FUNCTION_BLOCK EQ_StopperArm (* Servo that places the stopper; 0..180 degrees (outer home 120, inner 1), no feedback; equipment IO: owns its IO points, writes the output values its holder sends, reads its inputs every cycle and reports changes *)
  (* Standard: 61499-2 *)
  (* Version 0.1, 2026-09-28, Project contributors, AAU Smart Production Lab *)
  PACKAGE stoppering;
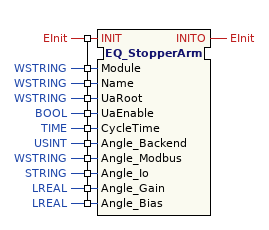
  EVENT_INPUT
    INIT : EInit WITH Module, Name, UaRoot, UaEnable, CycleTime, Angle_Backend, Angle_Modbus, Angle_Io, Angle_Gain, Angle_Bias;
  END_EVENT
  EVENT_OUTPUT
    INITO : EInit;
  END_EVENT
  VAR_INPUT
    Module : WSTRING;
    Name : WSTRING := "StopperArm";
    UaRoot : WSTRING;
    UaEnable : BOOL;
    CycleTime : TIME := T#50ms;
    Angle_Backend : USINT := 2;
    Angle_Modbus : WSTRING;
    Angle_Io : STRING;
    Angle_Gain : LREAL := 36.408;
    Angle_Bias : LREAL := 1638.4;
  END_VAR
  (* Group Core: One holder at a time, break before make, all off on release or abort; scanned every CycleTime *)
  (* Group Channels: Local channels to and from the skills (cmd, release, state), the module's state, and the inputs over OPC UA *)
  (* Group Outputs: The equipment's actuators: written on a change and every cycle, one block per IO point *)
  FBS
    Logic : stoppering::EL_StopperArm; {SET_ATTRIBUTE(GroupName, Core)}
    Cycle : iec61499::events::E_CYCLE; {SET_ATTRIBUTE(GroupName, Core)}
    Mode : modlib::MOD_StateView; {SET_ATTRIBUTE(GroupName, Channels)}
    SubCmd : iec61499::net::SUBSCRIBE_4(QI := TRUE); {SET_ATTRIBUTE(GroupName, Channels)}
    SubRelease : iec61499::net::SUBSCRIBE_1(QI := TRUE); {SET_ATTRIBUTE(GroupName, Channels)}
    PubState : iec61499::net::PUBLISH_1(QI := TRUE); {SET_ATTRIBUTE(GroupName, Channels)}
    Out_Angle : modlib::IO_AO; {SET_ATTRIBUTE(GroupName, Outputs)}
  END_FBS
  EVENT_CONNECTIONS
    INIT TO Logic.INIT;
    Logic.INITO TO Mode.INIT;
    Mode.INITO TO SubCmd.INIT;
    SubCmd.INITO TO SubRelease.INIT;
    SubRelease.INITO TO PubState.INIT;
    PubState.INITO TO Out_Angle.INIT;
    Out_Angle.INITO TO Cycle.START;
    Out_Angle.INITO TO INITO;
    SubCmd.IND TO Logic.CMD;
    SubRelease.IND TO Logic.RELEASE;
    Mode.CHG TO Logic.MOD_CHG;
    Cycle.EO TO Logic.REFRESH;
    Cycle.EO TO Logic.SAMPLE;
    Logic.STATE TO PubState.REQ;
    Logic.DRIVE TO Out_Angle.REQ;
    Out_Angle.CNF TO Logic.DRIVEN;
  END_CONNECTIONS
  DATA_CONNECTIONS
    Module TO Logic.Module;
    Name TO Logic.Name;
    Module TO Mode.Module;
    Logic.IdCmd TO SubCmd.ID;
    Logic.IdRelease TO SubRelease.ID;
    Logic.IdState TO PubState.ID;
    CycleTime TO Cycle.DT;
    SubCmd.RD_1 TO Logic.C_Holder;
    SubCmd.RD_2 TO Logic.C_Release;
    SubCmd.RD_3 TO Logic.C_Angle;
    SubCmd.RD_4 TO Logic.CE_Angle;
    SubRelease.RD_1 TO Logic.R_Holder;
    Mode.State TO Logic.ModState;
    Logic.Holder TO PubState.SD_1;
    Angle_Backend TO Out_Angle.Backend;
    Angle_Modbus TO Out_Angle.ModbusId;
    Angle_Io TO Out_Angle.IoName;
    Logic.O_Angle TO Out_Angle.OUT;
    Logic.E_Angle TO Out_Angle.EN;
    Angle_Gain TO Out_Angle.Gain;
    Angle_Bias TO Out_Angle.Bias;
  END_CONNECTIONS
END_FUNCTION_BLOCK
